FUNCTION_BLOCK SFC_COORD (* Basic Function Block Type *)
  (* Standard: 61499-2 *)
  (* Version 0.2, 2003-12-04, JHC, Rockwell Automation, Renamed for better indexing. *)
  (* Version 0.1, 2002-11-05, JHC, Rockwell Automation, Corrected missing ST element in Algorithm REQ. *)
  (* Version 0.0, 2000-05-30, JHC, Rockwell Automation *)
  (* Compiler header: package fb.rt.pnp; *)
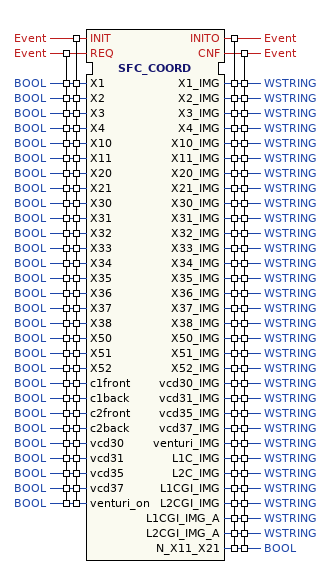
  EVENT_INPUT
    INIT WITH X1, X2, X3, X4, X30, X31, X32, X10, X11, X20, X21, c1front, c1back, c2front, c2back, X33, X34, X35, X36, X37, X38, vcd30, vcd31, vcd35, vcd37, venturi_on, X50, X51, X52; (* Initialization Request *)
    REQ WITH X1, X2, X3, X4, X30, X31, X32, c1front, c1back, c2front, X10, X11, X20, X21, c2back, X33, X34, X35, X36, X37, X38, vcd30, vcd31, vcd35, vcd37, venturi_on, X50, X51, X52; (* Normal Execution Request *)
  END_EVENT
  EVENT_OUTPUT
    INITO WITH X1_IMG, X2_IMG, X3_IMG, X4_IMG, vcd30_IMG, vcd31_IMG, vcd35_IMG, vcd37_IMG, venturi_IMG, X10_IMG, X11_IMG, X20_IMG, X21_IMG, L1C_IMG, L2C_IMG, X30_IMG, X31_IMG, X32_IMG, X33_IMG, X34_IMG, X35_IMG, X36_IMG, X37_IMG, X38_IMG, L1CGI_IMG, L2CGI_IMG, N_X11_X21, X50_IMG, X51_IMG, X52_IMG, L1CGI_IMG_A, L2CGI_IMG_A; (* Initialization Confirm *)
    CNF WITH X1_IMG, X2_IMG, X3_IMG, X4_IMG, vcd30_IMG, vcd31_IMG, vcd35_IMG, vcd37_IMG, venturi_IMG, X10_IMG, X11_IMG, X20_IMG, X21_IMG, L1C_IMG, L2C_IMG, X30_IMG, X31_IMG, X32_IMG, X33_IMG, X34_IMG, X35_IMG, X36_IMG, X37_IMG, X38_IMG, L1CGI_IMG, L2CGI_IMG, N_X11_X21, X50_IMG, X51_IMG, X52_IMG, L1CGI_IMG_A, L2CGI_IMG_A; (* Execution Confirmation *)
  END_EVENT
  VAR_INPUT
    X1 : BOOL; (* Input event qualifier *)
    X2 : BOOL;
    X3 : BOOL;
    X4 : BOOL;
    X10 : BOOL;
    X11 : BOOL;
    X20 : BOOL;
    X21 : BOOL;
    X30 : BOOL;
    X31 : BOOL;
    X32 : BOOL;
    X33 : BOOL;
    X34 : BOOL;
    X35 : BOOL;
    X36 : BOOL;
    X37 : BOOL;
    X38 : BOOL;
    X50 : BOOL;
    X51 : BOOL;
    X52 : BOOL;
    c1front : BOOL;
    c1back : BOOL;
    c2front : BOOL;
    c2back : BOOL;
    vcd30 : BOOL;
    vcd31 : BOOL;
    vcd35 : BOOL;
    vcd37 : BOOL;
    venturi_on : BOOL;
  END_VAR
  VAR_OUTPUT
    X1_IMG : WSTRING; (* Output event qualifier *)
    X2_IMG : WSTRING;
    X3_IMG : WSTRING;
    X4_IMG : WSTRING;
    X10_IMG : WSTRING;
    X11_IMG : WSTRING;
    X20_IMG : WSTRING;
    X21_IMG : WSTRING;
    X30_IMG : WSTRING;
    X31_IMG : WSTRING;
    X32_IMG : WSTRING;
    X33_IMG : WSTRING;
    X34_IMG : WSTRING;
    X35_IMG : WSTRING;
    X36_IMG : WSTRING;
    X37_IMG : WSTRING;
    X38_IMG : WSTRING;
    X50_IMG : WSTRING;
    X51_IMG : WSTRING;
    X52_IMG : WSTRING;
    vcd30_IMG : WSTRING;
    vcd31_IMG : WSTRING;
    vcd35_IMG : WSTRING;
    vcd37_IMG : WSTRING;
    venturi_IMG : WSTRING;
    L1C_IMG : WSTRING;
    L2C_IMG : WSTRING;
    L1CGI_IMG : WSTRING;
    L2CGI_IMG : WSTRING;
    L1CGI_IMG_A : WSTRING;
    L2CGI_IMG_A : WSTRING;
    N_X11_X21 : BOOL;
  END_VAR
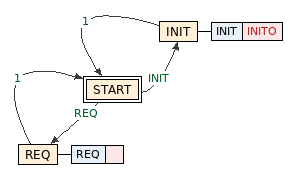
  EC_STATES
    START; (* Initial State *)
    INIT : INIT -> INITO; (* Initialization *)
    REQ : REQ; (* Normal execution *)
  END_STATES
  EC_TRANSITIONS
    START TO INIT := INIT;
    INIT TO START := 1;
    START TO REQ := REQ;
    REQ TO START := 1;
  END_TRANSITIONS
  ALGORITHM INIT IN ST: (* Initialization algorithm *)
X1_IMG := "/fb/rt/pnp/pics/S1.png";
X2_IMG := "/fb/rt/pnp/pics/S2.png";
X3_IMG := "/fb/rt/pnp/pics/S3.png";
X4_IMG := "/fb/rt/pnp/pics/S4.png";
X10_IMG := "/fb/rt/pnp/pics/S10.png";
X11_IMG := "/fb/rt/pnp/pics/S11.png";
X20_IMG := "/fb/rt/pnp/pics/S20.png";
X21_IMG := "/fb/rt/pnp/pics/S21.png";
X30_IMG := "/fb/rt/pnp/pics/S30.png";
X31_IMG := "/fb/rt/pnp/pics/S31.png";
X32_IMG := "/fb/rt/pnp/pics/S32.png";
X33_IMG := "/fb/rt/pnp/pics/S33.png";
X34_IMG := "/fb/rt/pnp/pics/S34.png";
X35_IMG := "/fb/rt/pnp/pics/S35.png";
X36_IMG := "/fb/rt/pnp/pics/S36.png";
X37_IMG := "/fb/rt/pnp/pics/S37.png";
X38_IMG := "/fb/rt/pnp/pics/S38.png";
X50_IMG := "/fb/rt/pnp/pics/S50.png";
X51_IMG := "/fb/rt/pnp/pics/S51.png";
X52_IMG := "/fb/rt/pnp/pics/S52.png";
vcd30_IMG := "/fb/rt/pnp/pics/VCGD.png";
vcd31_IMG := "/fb/rt/pnp/pics/VCGD.png";
vcd35_IMG := "/fb/rt/pnp/pics/VCGD.png";
vcd37_IMG := "/fb/rt/pnp/pics/VCGD.png";
venturi_IMG := "/fb/rt/pnp/pics/VENTURI.png";
L1C_IMG := "/fb/rt/pnp/pics/L1C.png";
L2C_IMG := "/fb/rt/pnp/pics/L2C.png";
L1CGI_IMG := "/fb/rt/pnp/pics/L1CGI.png";
L2CGI_IMG := "/fb/rt/pnp/pics/L2CGI.png";
L1CGI_IMG_A := "/fb/rt/pnp/pics/L1CGI.png";
L2CGI_IMG_A := "/fb/rt/pnp/pics/L2CGI.png";
N_X11_X21 := NOT (X11 OR X21);
  END_ALGORITHM
  ALGORITHM REQ IN ST: (* Normally executed algorithm *)
IF X1 THEN
IF X1_IMG = "/fb/rt/pnp/pics/S1.png" THEN
X1_IMG := "/fb/rt/pnp/pics/S1G.png";
CNF.serviceEvent(this);
END_IF
ELSE
IF X1_IMG = "/fb/rt/pnp/pics/S1G.png" THEN
X1_IMG := "/fb/rt/pnp/pics/S1.png";
CNF.serviceEvent(this);
END_IF
END_IF

IF X2 THEN
IF X2_IMG = "/fb/rt/pnp/pics/S2.png" THEN
X2_IMG := "/fb/rt/pnp/pics/S2G.png";
CNF.serviceEvent(this);
END_IF
ELSE
IF X2_IMG = "/fb/rt/pnp/pics/S2G.png" THEN
X2_IMG := "/fb/rt/pnp/pics/S2.png";
CNF.serviceEvent(this);
END_IF
END_IF

IF X3 THEN
IF X3_IMG = "/fb/rt/pnp/pics/S3.png" THEN
X3_IMG := "/fb/rt/pnp/pics/S3G.png";
CNF.serviceEvent(this);
END_IF
ELSE
IF X3_IMG = "/fb/rt/pnp/pics/S3G.png" THEN
X3_IMG := "/fb/rt/pnp/pics/S3.png";
CNF.serviceEvent(this);
END_IF
END_IF

IF X4 THEN
IF X4_IMG = "/fb/rt/pnp/pics/S4.png" THEN
X4_IMG := "/fb/rt/pnp/pics/S4G.png";
CNF.serviceEvent(this);
END_IF
ELSE
IF X4_IMG = "/fb/rt/pnp/pics/S4G.png" THEN
X4_IMG := "/fb/rt/pnp/pics/S4.png";
CNF.serviceEvent(this);
END_IF
END_IF

IF X10 THEN
IF X10_IMG = "/fb/rt/pnp/pics/S10.png" THEN
X10_IMG := "/fb/rt/pnp/pics/S10G.png";
CNF.serviceEvent(this);
END_IF
ELSE
IF X10_IMG = "/fb/rt/pnp/pics/S10G.png" THEN
X10_IMG := "/fb/rt/pnp/pics/S10.png";
CNF.serviceEvent(this);
END_IF
END_IF

IF X11 THEN
IF X11_IMG = "/fb/rt/pnp/pics/S11.png" THEN
X11_IMG := "/fb/rt/pnp/pics/S11G.png";
CNF.serviceEvent(this);
END_IF
ELSE
IF X11_IMG = "/fb/rt/pnp/pics/S11G.png" THEN
X11_IMG := "/fb/rt/pnp/pics/S11.png";
CNF.serviceEvent(this);
END_IF
END_IF

IF X20 THEN
IF X20_IMG = "/fb/rt/pnp/pics/S20.png" THEN
X20_IMG := "/fb/rt/pnp/pics/S20G.png";
CNF.serviceEvent(this);
END_IF
ELSE
IF X20_IMG = "/fb/rt/pnp/pics/S20G.png" THEN
X20_IMG := "/fb/rt/pnp/pics/S20.png";
CNF.serviceEvent(this);
END_IF
END_IF

IF X21 THEN
IF X21_IMG = "/fb/rt/pnp/pics/S21.png" THEN
X21_IMG := "/fb/rt/pnp/pics/S21G.png";
CNF.serviceEvent(this);
END_IF
ELSE
IF X21_IMG = "/fb/rt/pnp/pics/S21G.png" THEN
X21_IMG := "/fb/rt/pnp/pics/S21.png";
CNF.serviceEvent(this);
END_IF
END_IF

IF X30 THEN
IF X30_IMG = "/fb/rt/pnp/pics/S30.png" THEN
X30_IMG := "/fb/rt/pnp/pics/S30G.png";
CNF.serviceEvent(this);
END_IF
ELSE
IF X30_IMG = "/fb/rt/pnp/pics/S30G.png" THEN
X30_IMG := "/fb/rt/pnp/pics/S30.png";
CNF.serviceEvent(this);
END_IF
END_IF

IF X31 THEN
IF X31_IMG = "/fb/rt/pnp/pics/S31.png" THEN
X31_IMG := "/fb/rt/pnp/pics/S31G.png";
CNF.serviceEvent(this);
END_IF
ELSE
IF X31_IMG = "/fb/rt/pnp/pics/S31G.png" THEN
X31_IMG := "/fb/rt/pnp/pics/S31.png";
CNF.serviceEvent(this);
END_IF
END_IF

IF X32 THEN
IF X32_IMG = "/fb/rt/pnp/pics/S32.png" THEN
X32_IMG := "/fb/rt/pnp/pics/S32G.png";
CNF.serviceEvent(this);
END_IF
ELSE
IF X32_IMG = "/fb/rt/pnp/pics/S32G.png" THEN
X32_IMG := "/fb/rt/pnp/pics/S32.png";
CNF.serviceEvent(this);
END_IF
END_IF

IF X33 THEN
IF X33_IMG = "/fb/rt/pnp/pics/S33.png" THEN
X33_IMG := "/fb/rt/pnp/pics/S33G.png";
CNF.serviceEvent(this);
END_IF
ELSE
IF X33_IMG = "/fb/rt/pnp/pics/S33G.png" THEN
X33_IMG := "/fb/rt/pnp/pics/S33.png";
CNF.serviceEvent(this);
END_IF
END_IF

IF X34 THEN
IF X34_IMG = "/fb/rt/pnp/pics/S34.png" THEN
X34_IMG := "/fb/rt/pnp/pics/S34G.png";
CNF.serviceEvent(this);
END_IF
ELSE
IF X34_IMG = "/fb/rt/pnp/pics/S34G.png" THEN
X34_IMG := "/fb/rt/pnp/pics/S34.png";
CNF.serviceEvent(this);
END_IF
END_IF

IF X35 THEN
IF X35_IMG = "/fb/rt/pnp/pics/S35.png" THEN
X35_IMG := "/fb/rt/pnp/pics/S35G.png";
CNF.serviceEvent(this);
END_IF
ELSE
IF X35_IMG = "/fb/rt/pnp/pics/S35G.png" THEN
X35_IMG := "/fb/rt/pnp/pics/S35.png";
CNF.serviceEvent(this);
END_IF
END_IF

IF X36 THEN
IF X36_IMG = "/fb/rt/pnp/pics/S36.png" THEN
X36_IMG := "/fb/rt/pnp/pics/S36G.png";
CNF.serviceEvent(this);
END_IF
ELSE
IF X36_IMG = "/fb/rt/pnp/pics/S36G.png" THEN
X36_IMG := "/fb/rt/pnp/pics/S36.png";
CNF.serviceEvent(this);
END_IF
END_IF

IF X37 THEN
IF X37_IMG = "/fb/rt/pnp/pics/S37.png" THEN
X37_IMG := "/fb/rt/pnp/pics/S37G.png";
CNF.serviceEvent(this);
END_IF
ELSE
IF X37_IMG = "/fb/rt/pnp/pics/S37G.png" THEN
X37_IMG := "/fb/rt/pnp/pics/S37.png";
CNF.serviceEvent(this);
END_IF
END_IF

IF X38 THEN
IF X38_IMG = "/fb/rt/pnp/pics/S38.png" THEN
X38_IMG := "/fb/rt/pnp/pics/S38G.png";
CNF.serviceEvent(this);
END_IF
ELSE
IF X38_IMG = "/fb/rt/pnp/pics/S38G.png" THEN
X38_IMG := "/fb/rt/pnp/pics/S38.png";
CNF.serviceEvent(this);
END_IF
END_IF

IF X50 THEN
IF X50_IMG = "/fb/rt/pnp/pics/S50.png" THEN
X50_IMG := "/fb/rt/pnp/pics/S50G.png";
CNF.serviceEvent(this);
END_IF
ELSE
IF X50_IMG = "/fb/rt/pnp/pics/S50G.png" THEN
X50_IMG := "/fb/rt/pnp/pics/S50.png";
CNF.serviceEvent(this);
END_IF
END_IF

IF X51 THEN
IF X51_IMG = "/fb/rt/pnp/pics/S51.png" THEN
X51_IMG := "/fb/rt/pnp/pics/S51G.png";
CNF.serviceEvent(this);
END_IF
ELSE
IF X51_IMG = "/fb/rt/pnp/pics/S51G.png" THEN
X51_IMG := "/fb/rt/pnp/pics/S51.png";
CNF.serviceEvent(this);
END_IF
END_IF

IF X52 THEN
IF X52_IMG = "/fb/rt/pnp/pics/S52.png" THEN
X52_IMG := "/fb/rt/pnp/pics/S52G.png";
CNF.serviceEvent(this);
END_IF
ELSE
IF X52_IMG = "/fb/rt/pnp/pics/S52G.png" THEN
X52_IMG := "/fb/rt/pnp/pics/S52.png";
CNF.serviceEvent(this);
END_IF
END_IF

IF c1front THEN
IF L1C_IMG = "/fb/rt/pnp/pics/L1C.png" THEN
L1C_IMG := "/fb/rt/pnp/pics/L1CG.png";
CNF.serviceEvent(this);
END_IF
ELSE
IF L1C_IMG = "/fb/rt/pnp/pics/L1CG.png" THEN
L1C_IMG := "/fb/rt/pnp/pics/L1C.png";
CNF.serviceEvent(this);
END_IF
END_IF

IF c2front THEN
IF L2C_IMG = "/fb/rt/pnp/pics/L2C.png" THEN
L2C_IMG := "/fb/rt/pnp/pics/L2CG.png";
CNF.serviceEvent(this);
END_IF
ELSE
IF L2C_IMG = "/fb/rt/pnp/pics/L2CG.png" THEN
L2C_IMG := "/fb/rt/pnp/pics/L2C.png";
CNF.serviceEvent(this);
END_IF
END_IF

IF vcd30 THEN
IF vcd30_IMG = "/fb/rt/pnp/pics/VCGD.png" THEN
vcd30_IMG := "/fb/rt/pnp/pics/VCGDG.png";
CNF.serviceEvent(this);
END_IF
ELSE
IF vcd30_IMG = "/fb/rt/pnp/pics/VCGDG.png" THEN
vcd30_IMG := "/fb/rt/pnp/pics/VCGD.png";
CNF.serviceEvent(this);
END_IF
END_IF

IF vcd31 THEN
IF vcd31_IMG = "/fb/rt/pnp/pics/VCGD.png" THEN
vcd31_IMG := "/fb/rt/pnp/pics/VCGDG.png";
CNF.serviceEvent(this);
END_IF
ELSE
IF vcd31_IMG = "/fb/rt/pnp/pics/VCGDG.png" THEN
vcd31_IMG := "/fb/rt/pnp/pics/VCGD.png";
CNF.serviceEvent(this);
END_IF
END_IF

IF vcd35 THEN
IF vcd35_IMG = "/fb/rt/pnp/pics/VCGD.png" THEN
vcd35_IMG := "/fb/rt/pnp/pics/VCGDG.png";
CNF.serviceEvent(this);
END_IF
ELSE
IF vcd35_IMG = "/fb/rt/pnp/pics/VCGDG.png" THEN
vcd35_IMG := "/fb/rt/pnp/pics/VCGD.png";
CNF.serviceEvent(this);
END_IF
END_IF

IF vcd37 THEN
IF vcd37_IMG = "/fb/rt/pnp/pics/VCGD.png" THEN
vcd37_IMG := "/fb/rt/pnp/pics/VCGDG.png";
CNF.serviceEvent(this);
END_IF
ELSE
IF vcd37_IMG = "/fb/rt/pnp/pics/VCGDG.png" THEN
vcd37_IMG := "/fb/rt/pnp/pics/VCGD.png";
CNF.serviceEvent(this);
END_IF
END_IF

IF venturi_on THEN
IF venturi_IMG = "/fb/rt/pnp/pics/VENTURI.png" THEN
venturi_IMG := "/fb/rt/pnp/pics/VENTURIG.png";
CNF.serviceEvent(this);
END_IF
ELSE
IF venturi_IMG = "/fb/rt/pnp/pics/VENTURIG.png" THEN
venturi_IMG := "/fb/rt/pnp/pics/VENTURI.png";
CNF.serviceEvent(this);
END_IF
END_IF

IF c1back & X33 THEN
IF L1CGI_IMG = "/fb/rt/pnp/pics/L1CGI.png" THEN
L1CGI_IMG := "/fb/rt/pnp/pics/L1CGIG.png";
CNF.serviceEvent(this);
END_IF
ELSE
IF L1CGI_IMG = "/fb/rt/pnp/pics/L1CGIG.png" THEN
L1CGI_IMG := "/fb/rt/pnp/pics/L1CGI.png";
CNF.serviceEvent(this);
END_IF
END_IF

IF c2back & X34 THEN
IF L2CGI_IMG = "/fb/rt/pnp/pics/L2CGI.png" THEN
L2CGI_IMG := "/fb/rt/pnp/pics/L2CGIG.png";
CNF.serviceEvent(this);
END_IF
ELSE
IF L2CGI_IMG = "/fb/rt/pnp/pics/L2CGIG.png" THEN
L2CGI_IMG := "/fb/rt/pnp/pics/L2CGI.png";
CNF.serviceEvent(this);
END_IF
END_IF

IF c1back & X51 THEN
IF L1CGI_IMG_A = "/fb/rt/pnp/pics/L1CGI.png" THEN
L1CGI_IMG_A := "/fb/rt/pnp/pics/L1CGIG.png";
CNF.serviceEvent(this);
END_IF
ELSE
IF L1CGI_IMG_A = "/fb/rt/pnp/pics/L1CGIG.png" THEN
L1CGI_IMG_A := "/fb/rt/pnp/pics/L1CGI.png";
CNF.serviceEvent(this);
END_IF
END_IF

IF c2back & X52 THEN
IF L2CGI_IMG_A = "/fb/rt/pnp/pics/L2CGI.png" THEN
L2CGI_IMG_A := "/fb/rt/pnp/pics/L2CGIG.png";
CNF.serviceEvent(this);
END_IF
ELSE
IF L2CGI_IMG_A = "/fb/rt/pnp/pics/L2CGIG.png" THEN
L2CGI_IMG_A := "/fb/rt/pnp/pics/L2CGI.png";
CNF.serviceEvent(this);
END_IF
END_IF

N_X11_X21 := NOT (X11 OR X21);
  END_ALGORITHM
END_FUNCTION_BLOCK
